Yaskawa INFORM job: R2_O1(45,180).JBI

/JOB
//NAME R2_O1(45,180)
///FOLDERNAME PROGRAMY_TESTOWE_ODWLOK
//POS
///NPOS 26,26,26,2,0,0
///TOOL 0
///POSTYPE PULSE
///PULSE
C00000=-126255,-92505,-103564,60413,100364,46248
C00001=-126224,-93141,-87205,58847,94872,42094
C00002=-122946,-92654,-83603,58597,91802,41922
C00003=-121632,-92322,-82104,58529,90589,41869
C00004=-119348,-92327,-82111,58462,89189,42288
C00005=-121632,-92322,-82104,58529,90589,41869
C00006=-125857,-95605,-78941,58367,91212,39674
C00007=-125974,-97624,-78508,58308,90574,39144
C00008=-125857,-95605,-78941,58367,91212,39674
C00009=-126085,-103168,-90405,58557,93070,40869
C00010=-110885,-104078,-90031,58087,83374,43399
C00011=-111093,-100811,-87655,58084,83619,43444
C00012=-110885,-104078,-90031,58087,83374,43399
C00013=-126085,-103168,-90405,58557,93070,40869
C00014=-121632,-92322,-82104,58529,90589,41869
C00015=-122946,-92654,-83603,58597,91802,41922
C00016=-126224,-93141,-87205,58847,94872,42094
C00017=-126255,-92505,-103564,60413,100364,46248
C00018=-120633,-97999,-84570,33805,55883,32041
C00019=-120634,-97982,-84564,33804,55888,32042
C00020=-120635,-97975,-84561,33803,55890,32042
C00021=-120639,-98412,-85985,33568,56438,32236
C00022=-120641,-100925,-85907,34063,55317,31832
C00023=-120635,-97890,-84529,33794,55910,32050
C00024=-120634,-97897,-84532,33795,55908,32049
C00025=-120633,-97913,-84538,33796,55903,32048
BC00000=284759,739774,628289
BC00001=284759,739774,628289
BC00002=284759,739774,628289
BC00003=284759,739774,628289
BC00004=284759,739774,628289
BC00005=284759,739774,628289
BC00006=284759,739774,628289
BC00007=284759,739774,628289
BC00008=284759,739774,628289
BC00009=284759,739774,628289
BC00010=284759,739774,628289
BC00011=284759,739774,628289
BC00012=284759,739774,628289
BC00013=284759,739774,628289
BC00014=284759,739774,628289
BC00015=284759,739774,628289
BC00016=284759,739774,628289
BC00017=284759,739774,628289
BC00018=332447,660018,685021
BC00019=333175,664889,664382
BC00020=333466,666838,656127
BC00021=333466,666838,656127
BC00022=333466,666838,656127
BC00023=355140,666762,656312
BC00024=354849,664813,664568
BC00025=354121,659942,685206
EC00000=399078,1112951
EC00001=399078,1112951
EC00002=399078,1112951
EC00003=399078,1112951
EC00004=399078,1112951
EC00005=399078,1112951
EC00006=399078,1112951
EC00007=399078,1112951
EC00008=399078,1112951
EC00009=399078,1112951
EC00010=399078,1112951
EC00011=399078,1112951
EC00012=399078,1112951
EC00013=399078,1112951
EC00014=399078,1112951
EC00015=399078,1112951
EC00016=399078,1112951
EC00017=399078,1112951
EC00018=399078,1112951
EC00019=399078,1112951
EC00020=399078,1112951
EC00021=399078,1112951
EC00022=399078,1112951
EC00023=399078,1112951
EC00024=399078,1112951
EC00025=399078,1112951
///POSTYPE BASE
///RECTAN
///RCONF 0,0,0,0,0,0,0,0,0,0,0,0,0,0,0,0,0,0,0,0,0,0,0,0
P00006=0.222,-3.123,-1.508,0.0000,0.0000,0.0000
P00021=-0.225,-6.128,-0.405,0.0000,0.0000,0.0000
//INST
///DATE 2023/11/22 16:04
///ATTR SC,RW
///GROUP1 RB1,BS1
///GROUP2 ST1
NOP
'r2_O1(45,180)
'Path S1189
SSFTOF
MOVJ C00000 BC00000 VJ=100.00  +MOVJ EC00000 VJ=100.00
MOVJ C00001 BC00001 VJ=100.00  +MOVJ EC00001 VJ=100.00
MOVL C00002 BC00002 V=400.0  +MOVJ EC00002 VJ=100.00
SMOVL C00003 BC00003 V=60.0  +MOVJ EC00003
SREFP 3 C00004 BC00004  +REFP EC00004
CALL JOB:SEARCH-R1-S1
SET P021 P006
SSFTON P021
SMOVL C00005 BC00005 V=60.0  +MOVJ EC00005
SMOVL C00006 BC00006 V=60.0  +MOVJ EC00006
SREFP 3 C00007 BC00007  +REFP EC00007
CALL JOB:SEARCH-R1-S1
SET P021 P006
SSFTON P021
SMOVL C00008 BC00008 V=60.0  +MOVJ EC00008
SMOVL C00009 BC00009 V=100.0  +MOVJ EC00009
SMOVL C00010 BC00010 V=60.0  +MOVJ EC00010
SREFP 3 C00011 BC00011  +REFP EC00011
CALL JOB:SEARCH-R1-S1
SET P021 P006
SSFTON P021
SMOVL C00012 BC00012 V=60.0  +MOVJ EC00012
SMOVL C00013 BC00013 V=100.0  +MOVJ EC00013
SMOVL C00014 BC00014 V=100.0  +MOVJ EC00014
MOVL C00015 BC00015 V=400.0  +MOVJ EC00015 VJ=100.00
MOVL C00016 BC00016 V=1000.0  +MOVJ EC00016 VJ=100.00
MOVL C00017 BC00017 V=1000.0  +MOVJ EC00017 VJ=100.00
'Path W1190
SSFTOF
SSFTON P021
MOVJ C00018 BC00018 VJ=100.00  +MOVJ EC00018 VJ=100.00
SMOVL C00019 BC00019 V=400.0  +MOVJ EC00019
SMOVL C00020 BC00020 V=100.0 PL=0  +MOVJ EC00020
SREFP 1 C00021 BC00021  +REFP EC00021
SREFP 2 C00022 BC00022  +REFP EC00022
MACRO1 MJ#(0) ARGF0
ARCON
SMOVL C00023 BC00023 V=10.0  +MOVJ EC00023
ARCOF
SMOVL C00024 BC00024 V=400.0  +MOVJ EC00024
SMOVL C00025 BC00025 V=1000.0  +MOVJ EC00025
SSFTOF
END
